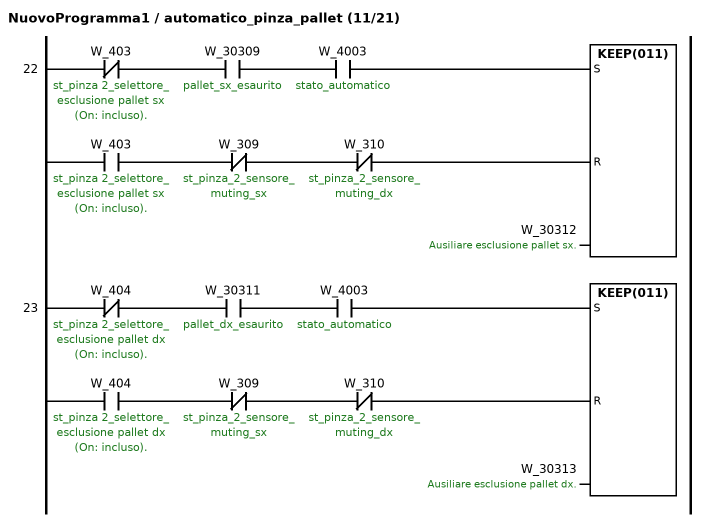
; [picture p72: NuovoProgramma1 / automatico_pinza_pallet, rungs 22-23]
; rung 22
LDNOT W_403  ; st_pinza 2_selettore_esclusione pallet sx (On: incluso).
AND W_30309  ; pallet_sx_esaurito
AND W_4003  ; stato_automatico
LD W_403  ; st_pinza 2_selettore_esclusione pallet sx (On: incluso).
ANDNOT W_309  ; st_pinza_2_sensore_muting_sx
ANDNOT W_310  ; st_pinza_2_sensore_muting_dx
KEEP(011) W_30312  ; Ausiliare esclusione pallet sx.
; rung 23
LDNOT W_404  ; st_pinza 2_selettore_esclusione pallet dx (On: incluso).
AND W_30311  ; pallet_dx_esaurito
AND W_4003  ; stato_automatico
LD W_404  ; st_pinza 2_selettore_esclusione pallet dx (On: incluso).
ANDNOT W_309  ; st_pinza_2_sensore_muting_sx
ANDNOT W_310  ; st_pinza_2_sensore_muting_dx
KEEP(011) W_30313  ; Ausiliare esclusione pallet dx.

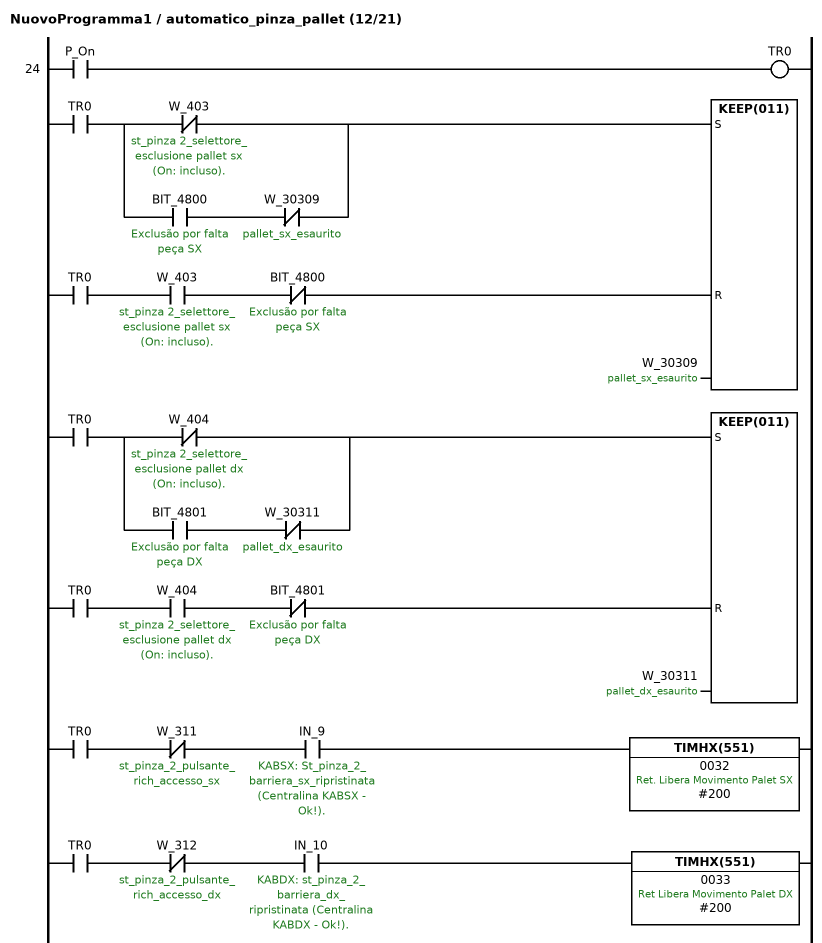

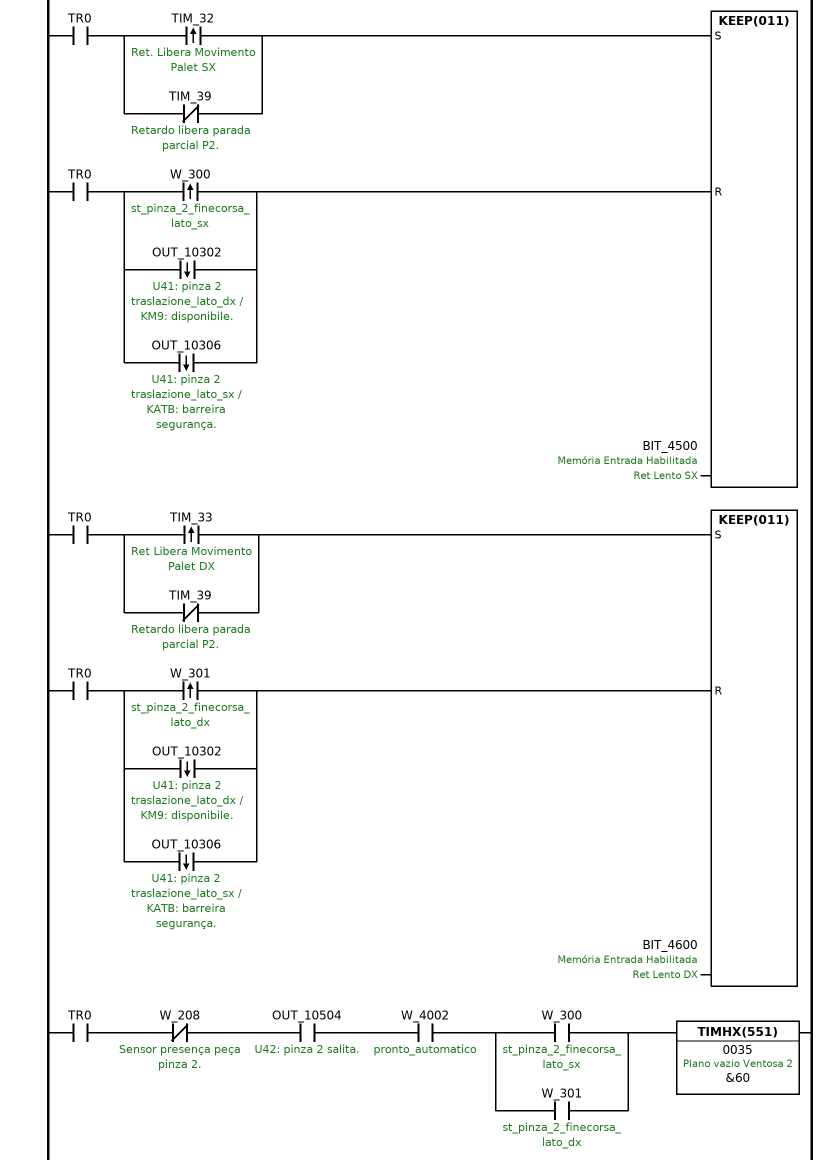

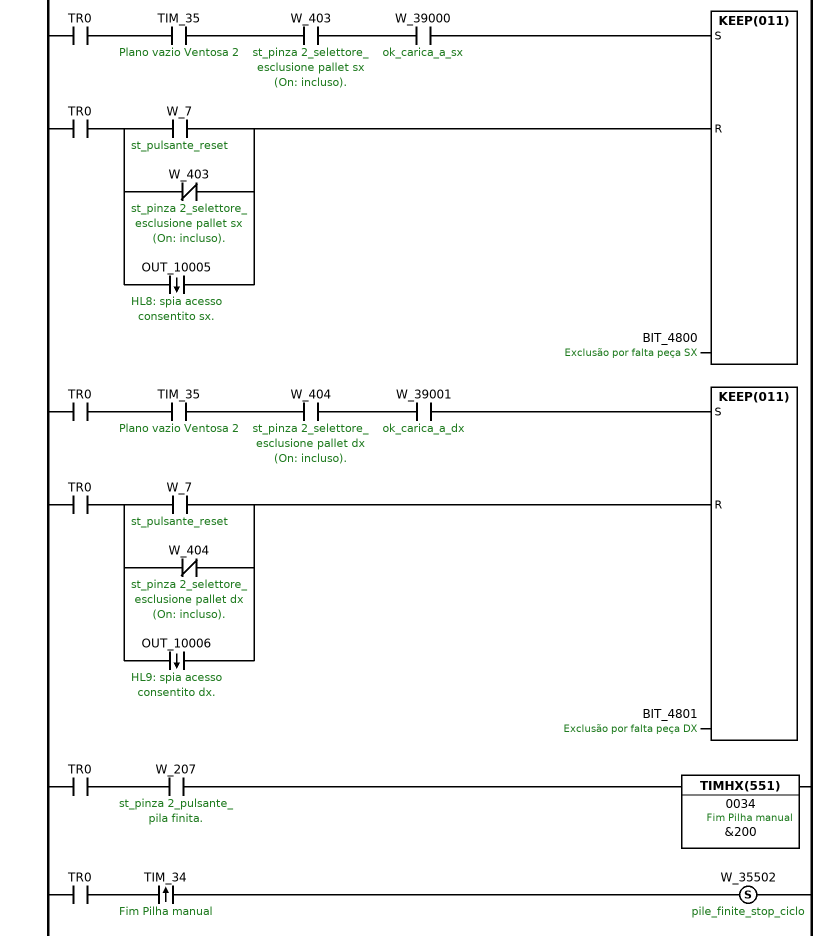
; rung 24
LD P_On
OUT TR0
LDNOT W_403  ; st_pinza 2_selettore_esclusione pallet sx (On: incluso).
LD BIT_4800  ; Exclusão por falta peça SX
ANDNOT W_30309  ; pallet_sx_esaurito
ORLD
ANDLD
LD TR0
AND W_403  ; st_pinza 2_selettore_esclusione pallet sx (On: incluso).
ANDNOT BIT_4800  ; Exclusão por falta peça SX
KEEP(011) W_30309  ; pallet_sx_esaurito
LD TR0
LDNOT W_404  ; st_pinza 2_selettore_esclusione pallet dx (On: incluso).
LD BIT_4801  ; Exclusão por falta peça DX
ANDNOT W_30311  ; pallet_dx_esaurito
ORLD
ANDLD
LD TR0
AND W_404  ; st_pinza 2_selettore_esclusione pallet dx (On: incluso).
ANDNOT BIT_4801  ; Exclusão por falta peça DX
KEEP(011) W_30311  ; pallet_dx_esaurito
LD TR0
ANDNOT W_311  ; st_pinza_2_pulsante_rich_accesso_sx
AND IN_9  ; KABSX: St_pinza_2_barriera_sx_ripristinata (Centralina KABSX - Ok!).
TIMHX(551) 0032 #200  ; Ret. Libera Movimento Palet SX
LD TR0
ANDNOT W_312  ; st_pinza_2_pulsante_rich_accesso_dx
AND IN_10  ; KABDX: st_pinza_2_barriera_dx_ripristinata (Centralina KABDX - Ok!).
TIMHX(551) 0033 #200  ; Ret Libera Movimento Palet DX
LD TR0
@LD TIM_32  ; Ret. Libera Movimento Palet SX
ORNOT TIM_39  ; Retardo libera parada parcial P2.
ANDLD
LD TR0
@LD W_300  ; st_pinza_2_finecorsa_lato_sx
%OR OUT_10302  ; U41: pinza 2 traslazione_lato_dx / KM9: disponibile.
%OR OUT_10306  ; U41: pinza 2 traslazione_lato_sx / KATB: barreira segurança.
ANDLD
KEEP(011) BIT_4500  ; Memória Entrada Habilitada Ret Lento SX
LD TR0
@LD TIM_33  ; Ret Libera Movimento Palet DX
ORNOT TIM_39  ; Retardo libera parada parcial P2.
ANDLD
LD TR0
@LD W_301  ; st_pinza_2_finecorsa_lato_dx
%OR OUT_10302  ; U41: pinza 2 traslazione_lato_dx / KM9: disponibile.
%OR OUT_10306  ; U41: pinza 2 traslazione_lato_sx / KATB: barreira segurança.
ANDLD
KEEP(011) BIT_4600  ; Memória Entrada Habilitada Ret Lento DX
LD TR0
ANDNOT W_208  ; Sensor presença peça pinza 2.
AND OUT_10504  ; U42: pinza 2 salita.
AND W_4002  ; pronto_automatico
LD W_300  ; st_pinza_2_finecorsa_lato_sx
OR W_301  ; st_pinza_2_finecorsa_lato_dx
ANDLD
TIMHX(551) 0035 &60  ; Plano vazio Ventosa 2
LD TR0
AND TIM_35  ; Plano vazio Ventosa 2
AND W_403  ; st_pinza 2_selettore_esclusione pallet sx (On: incluso).
AND W_39000  ; ok_carica_a_sx
LD TR0
LD W_7  ; st_pulsante_reset
ORNOT W_403  ; st_pinza 2_selettore_esclusione pallet sx (On: incluso).
%OR OUT_10005  ; HL8: spia acesso consentito sx.
ANDLD
KEEP(011) BIT_4800  ; Exclusão por falta peça SX
LD TR0
AND TIM_35  ; Plano vazio Ventosa 2
AND W_404  ; st_pinza 2_selettore_esclusione pallet dx (On: incluso).
AND W_39001  ; ok_carica_a_dx
LD TR0
LD W_7  ; st_pulsante_reset
ORNOT W_404  ; st_pinza 2_selettore_esclusione pallet dx (On: incluso).
%OR OUT_10006  ; HL9: spia acesso consentito dx.
ANDLD
KEEP(011) BIT_4801  ; Exclusão por falta peça DX
LD TR0
AND W_207  ; st_pinza 2_pulsante_pila finita.
TIMHX(551) 0034 &200  ; Fim Pilha manual
LD TR0
@AND TIM_34  ; Fim Pilha manual
SET W_35502  ; pile_finite_stop_ciclo

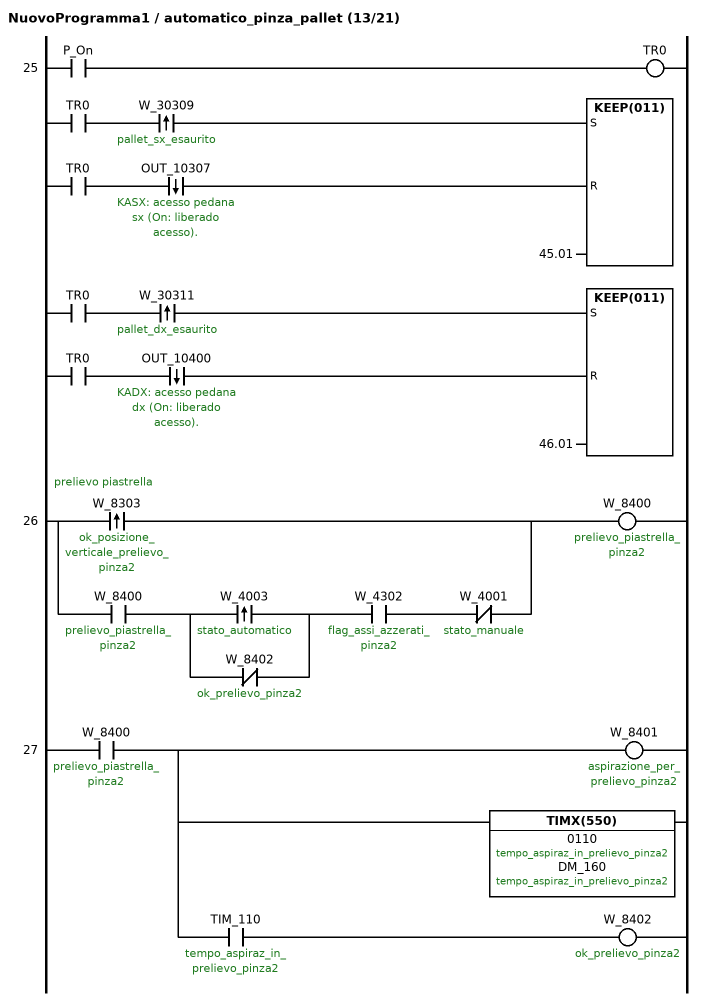
; rung 25
LD P_On
OUT TR0
@AND W_30309  ; pallet_sx_esaurito
LD TR0
%AND OUT_10307  ; KASX: acesso pedana sx (On: liberado acesso).
KEEP(011) 45.01
LD TR0
@AND W_30311  ; pallet_dx_esaurito
LD TR0
%AND OUT_10400  ; KADX: acesso pedana dx (On: liberado acesso).
KEEP(011) 46.01
; rung 26: prelievo piastrella
@LD W_8303  ; ok_posizione_verticale_prelievo_pinza2
LD W_8400  ; prelievo_piastrella_pinza2
@LD W_4003  ; stato_automatico
ORNOT W_8402  ; ok_prelievo_pinza2
ANDLD
AND W_4302  ; flag_assi_azzerati_pinza2
ANDNOT W_4001  ; stato_manuale
ORLD
OUT W_8400  ; prelievo_piastrella_pinza2
; rung 27
LD W_8400  ; prelievo_piastrella_pinza2
OUT W_8401  ; aspirazione_per_prelievo_pinza2
TIMX(550) 0110 DM_160  ; tempo_aspiraz_in_prelievo_pinza2
AND TIM_110  ; tempo_aspiraz_in_prelievo_pinza2
OUT W_8402  ; ok_prelievo_pinza2

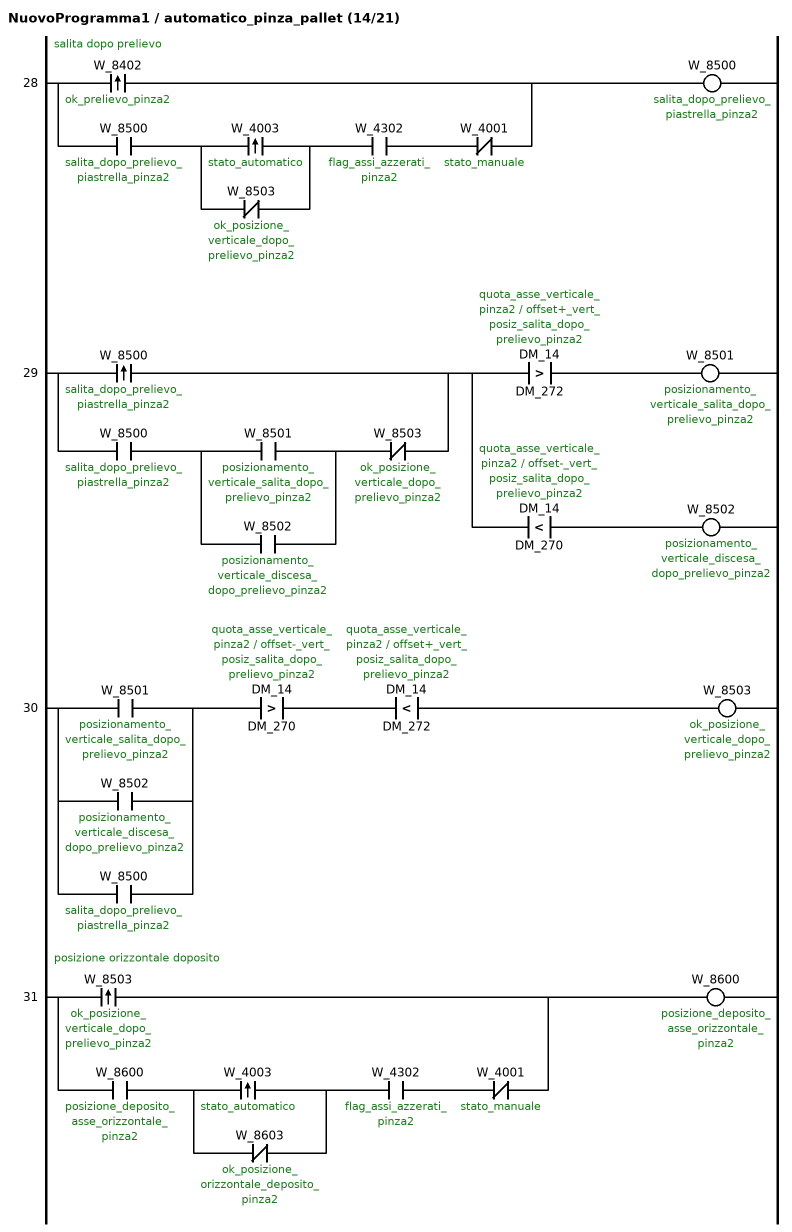
; rung 28: salita dopo prelievo
@LD W_8402  ; ok_prelievo_pinza2
LD W_8500  ; salita_dopo_prelievo_piastrella_pinza2
@LD W_4003  ; stato_automatico
ORNOT W_8503  ; ok_posizione_verticale_dopo_prelievo_pinza2
ANDLD
AND W_4302  ; flag_assi_azzerati_pinza2
ANDNOT W_4001  ; stato_manuale
ORLD
OUT W_8500  ; salita_dopo_prelievo_piastrella_pinza2
; rung 29
@LD W_8500  ; salita_dopo_prelievo_piastrella_pinza2
LD W_8500  ; salita_dopo_prelievo_piastrella_pinza2
LD W_8501  ; posizionamento_verticale_salita_dopo_prelievo_pinza2
OR W_8502  ; posizionamento_verticale_discesa_dopo_prelievo_pinza2
ANDLD
ANDNOT W_8503  ; ok_posizione_verticale_dopo_prelievo_pinza2
ORLD
OUT TR0
AND>SL(323) DM_14 DM_272  ; quota_asse_verticale_pinza2, offset+_vert_posiz_salita_dopo_prelievo_pinza2
OUT W_8501  ; posizionamento_verticale_salita_dopo_prelievo_pinza2
LD TR0
AND<SL(313) DM_14 DM_270  ; quota_asse_verticale_pinza2, offset-_vert_posiz_salita_dopo_prelievo_pinza2
OUT W_8502  ; posizionamento_verticale_discesa_dopo_prelievo_pinza2
; rung 30
LD W_8501  ; posizionamento_verticale_salita_dopo_prelievo_pinza2
OR W_8502  ; posizionamento_verticale_discesa_dopo_prelievo_pinza2
OR W_8500  ; salita_dopo_prelievo_piastrella_pinza2
AND>SL(323) DM_14 DM_270  ; quota_asse_verticale_pinza2, offset-_vert_posiz_salita_dopo_prelievo_pinza2
AND<SL(313) DM_14 DM_272  ; quota_asse_verticale_pinza2, offset+_vert_posiz_salita_dopo_prelievo_pinza2
OUT W_8503  ; ok_posizione_verticale_dopo_prelievo_pinza2
; rung 31: posizione orizzontale doposito
@LD W_8503  ; ok_posizione_verticale_dopo_prelievo_pinza2
LD W_8600  ; posizione_deposito_asse_orizzontale_pinza2
@LD W_4003  ; stato_automatico
ORNOT W_8603  ; ok_posizione_orizzontale_deposito_pinza2
ANDLD
AND W_4302  ; flag_assi_azzerati_pinza2
ANDNOT W_4001  ; stato_manuale
ORLD
OUT W_8600  ; posizione_deposito_asse_orizzontale_pinza2

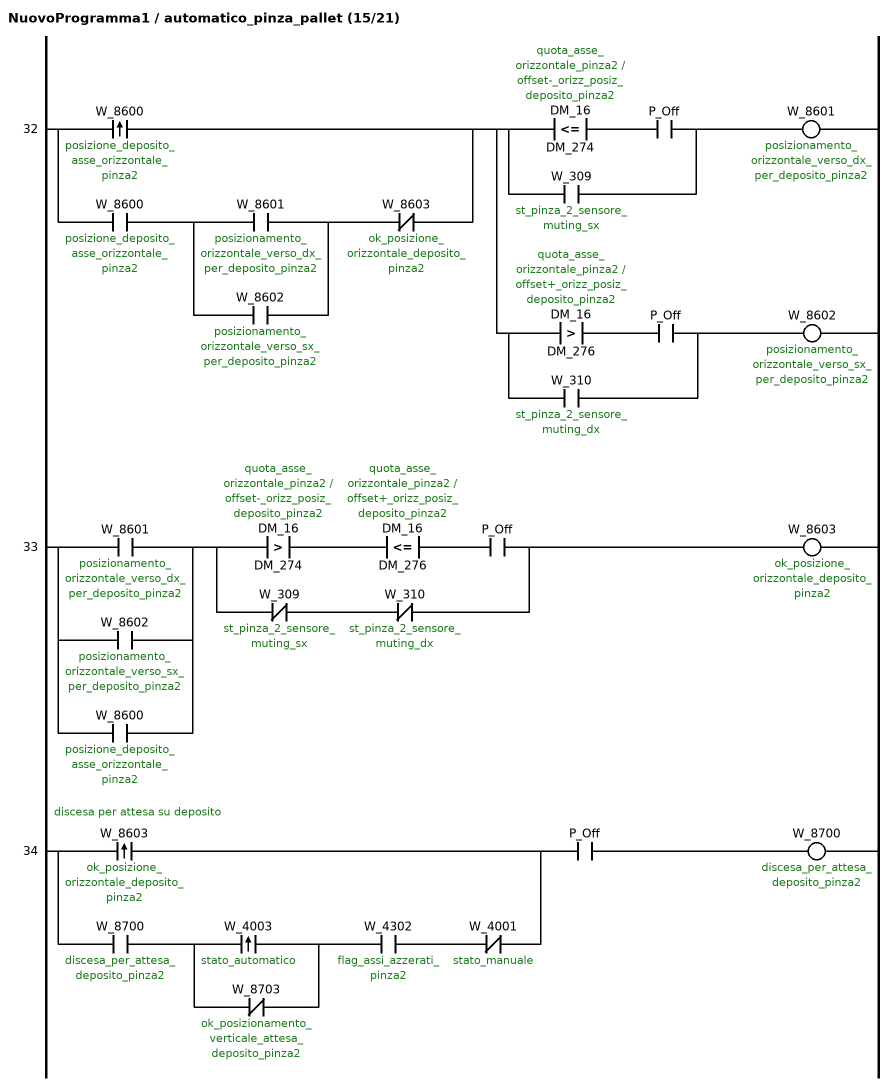
; rung 32
@LD W_8600  ; posizione_deposito_asse_orizzontale_pinza2
LD W_8600  ; posizione_deposito_asse_orizzontale_pinza2
LD W_8601  ; posizionamento_orizzontale_verso_dx_per_deposito_pinza2
OR W_8602  ; posizionamento_orizzontale_verso_sx_per_deposito_pinza2
ANDLD
ANDNOT W_8603  ; ok_posizione_orizzontale_deposito_pinza2
ORLD
OUT TR0
LD<=SL(318) DM_16 DM_274  ; quota_asse_orizzontale_pinza2, offset-_orizz_posiz_deposito_pinza2
AND P_Off
OR W_309  ; st_pinza_2_sensore_muting_sx
ANDLD
OUT W_8601  ; posizionamento_orizzontale_verso_dx_per_deposito_pinza2
LD TR0
LD>SL(323) DM_16 DM_276  ; quota_asse_orizzontale_pinza2, offset+_orizz_posiz_deposito_pinza2
AND P_Off
OR W_310  ; st_pinza_2_sensore_muting_dx
ANDLD
OUT W_8602  ; posizionamento_orizzontale_verso_sx_per_deposito_pinza2
; rung 33
LD W_8601  ; posizionamento_orizzontale_verso_dx_per_deposito_pinza2
OR W_8602  ; posizionamento_orizzontale_verso_sx_per_deposito_pinza2
OR W_8600  ; posizione_deposito_asse_orizzontale_pinza2
LD>SL(323) DM_16 DM_274  ; quota_asse_orizzontale_pinza2, offset-_orizz_posiz_deposito_pinza2
AND<=SL(318) DM_16 DM_276  ; quota_asse_orizzontale_pinza2, offset+_orizz_posiz_deposito_pinza2
AND P_Off
LDNOT W_309  ; st_pinza_2_sensore_muting_sx
ANDNOT W_310  ; st_pinza_2_sensore_muting_dx
ORLD
ANDLD
OUT W_8603  ; ok_posizione_orizzontale_deposito_pinza2
; rung 34: discesa per attesa su deposito
@LD W_8603  ; ok_posizione_orizzontale_deposito_pinza2
LD W_8700  ; discesa_per_attesa_deposito_pinza2
@LD W_4003  ; stato_automatico
ORNOT W_8703  ; ok_posizionamento_verticale_attesa_deposito_pinza2
ANDLD
AND W_4302  ; flag_assi_azzerati_pinza2
ANDNOT W_4001  ; stato_manuale
ORLD
AND P_Off
OUT W_8700  ; discesa_per_attesa_deposito_pinza2

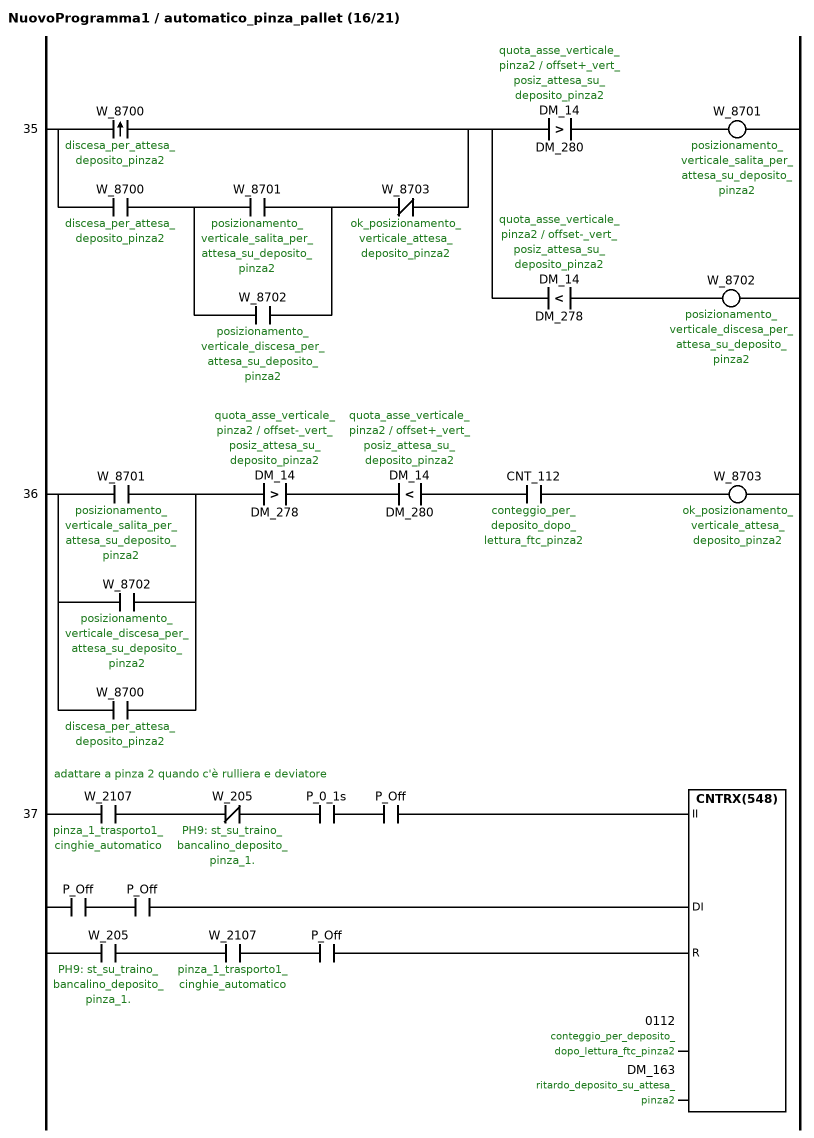
; rung 35
@LD W_8700  ; discesa_per_attesa_deposito_pinza2
LD W_8700  ; discesa_per_attesa_deposito_pinza2
LD W_8701  ; posizionamento_verticale_salita_per_attesa_su_deposito_pinza2
OR W_8702  ; posizionamento_verticale_discesa_per_attesa_su_deposito_pinza2
ANDLD
ANDNOT W_8703  ; ok_posizionamento_verticale_attesa_deposito_pinza2
ORLD
OUT TR0
AND>SL(323) DM_14 DM_280  ; quota_asse_verticale_pinza2, offset+_vert_posiz_attesa_su_deposito_pinza2
OUT W_8701  ; posizionamento_verticale_salita_per_attesa_su_deposito_pinza2
LD TR0
AND<SL(313) DM_14 DM_278  ; quota_asse_verticale_pinza2, offset-_vert_posiz_attesa_su_deposito_pinza2
OUT W_8702  ; posizionamento_verticale_discesa_per_attesa_su_deposito_pinza2
; rung 36
LD W_8701  ; posizionamento_verticale_salita_per_attesa_su_deposito_pinza2
OR W_8702  ; posizionamento_verticale_discesa_per_attesa_su_deposito_pinza2
OR W_8700  ; discesa_per_attesa_deposito_pinza2
AND>SL(323) DM_14 DM_278  ; quota_asse_verticale_pinza2, offset-_vert_posiz_attesa_su_deposito_pinza2
AND<SL(313) DM_14 DM_280  ; quota_asse_verticale_pinza2, offset+_vert_posiz_attesa_su_deposito_pinza2
AND CNT_112  ; conteggio_per_deposito_dopo_lettura_ftc_pinza2
OUT W_8703  ; ok_posizionamento_verticale_attesa_deposito_pinza2
; rung 37: adattare a pinza 2 quando c'è rulliera e deviatore
LD W_2107  ; pinza_1_trasporto1_cinghie_automatico
ANDNOT W_205  ; PH9: st_su_traino_bancalino_deposito_pinza_1.
AND P_0_1s
AND P_Off
LD P_Off
AND P_Off
LD W_205  ; PH9: st_su_traino_bancalino_deposito_pinza_1.
AND W_2107  ; pinza_1_trasporto1_cinghie_automatico
AND P_Off
CNTRX(548) 0112 DM_163  ; ritardo_deposito_su_attesa_pinza2, conteggio_per_deposito_dopo_lettura_ftc_pinza2

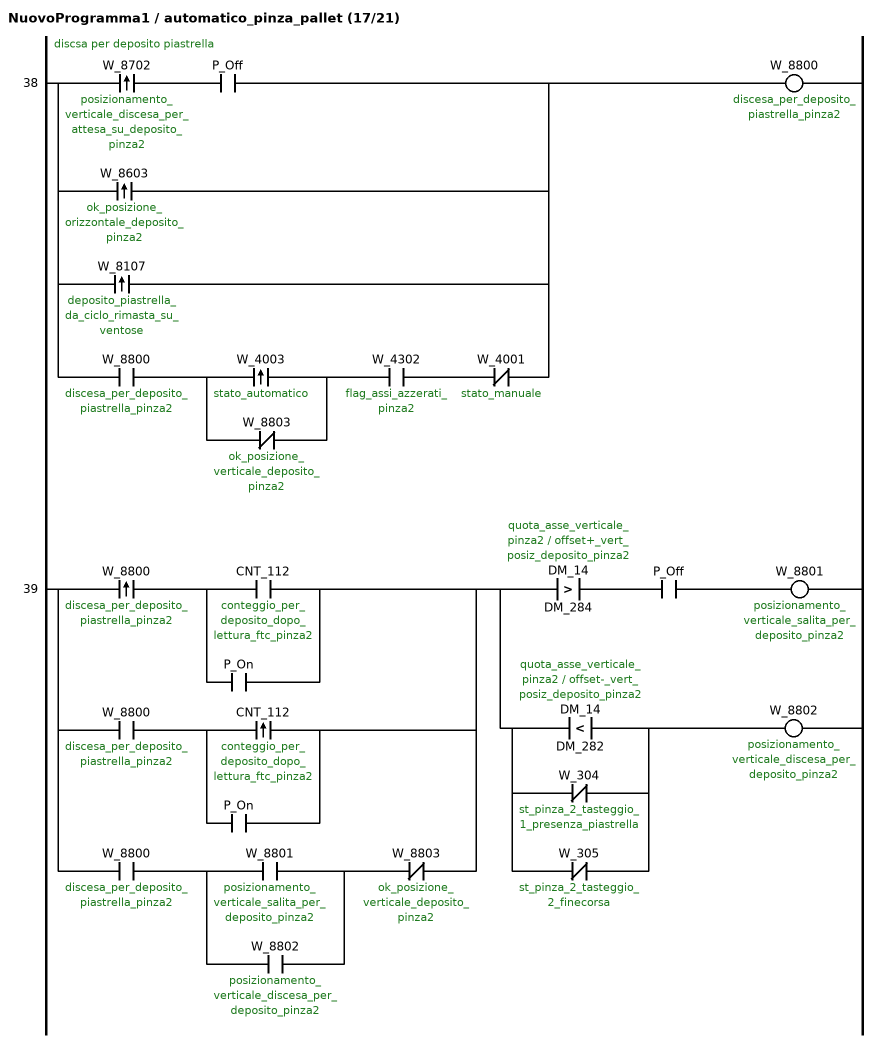
; rung 38: discsa per deposito piastrella
@LD W_8702  ; posizionamento_verticale_discesa_per_attesa_su_deposito_pinza2
AND P_Off
@OR W_8603  ; ok_posizione_orizzontale_deposito_pinza2
@OR W_8107  ; deposito_piastrella_da_ciclo_rimasta_su_ventose
LD W_8800  ; discesa_per_deposito_piastrella_pinza2
@LD W_4003  ; stato_automatico
ORNOT W_8803  ; ok_posizione_verticale_deposito_pinza2
ANDLD
AND W_4302  ; flag_assi_azzerati_pinza2
ANDNOT W_4001  ; stato_manuale
ORLD
OUT W_8800  ; discesa_per_deposito_piastrella_pinza2
; rung 39
@LD W_8800  ; discesa_per_deposito_piastrella_pinza2
LD CNT_112  ; conteggio_per_deposito_dopo_lettura_ftc_pinza2
OR P_On
ANDLD
LD W_8800  ; discesa_per_deposito_piastrella_pinza2
@LD CNT_112  ; conteggio_per_deposito_dopo_lettura_ftc_pinza2
OR P_On
ANDLD
ORLD
LD W_8800  ; discesa_per_deposito_piastrella_pinza2
LD W_8801  ; posizionamento_verticale_salita_per_deposito_pinza2
OR W_8802  ; posizionamento_verticale_discesa_per_deposito_pinza2
ANDLD
ANDNOT W_8803  ; ok_posizione_verticale_deposito_pinza2
ORLD
OUT TR0
AND>SL(323) DM_14 DM_284  ; quota_asse_verticale_pinza2, offset+_vert_posiz_deposito_pinza2
AND P_Off
OUT W_8801  ; posizionamento_verticale_salita_per_deposito_pinza2
LD TR0
LD<SL(313) DM_14 DM_282  ; quota_asse_verticale_pinza2, offset-_vert_posiz_deposito_pinza2
ORNOT W_304  ; st_pinza_2_tasteggio_1_presenza_piastrella
ORNOT W_305  ; st_pinza_2_tasteggio_2_finecorsa
ANDLD
OUT W_8802  ; posizionamento_verticale_discesa_per_deposito_pinza2

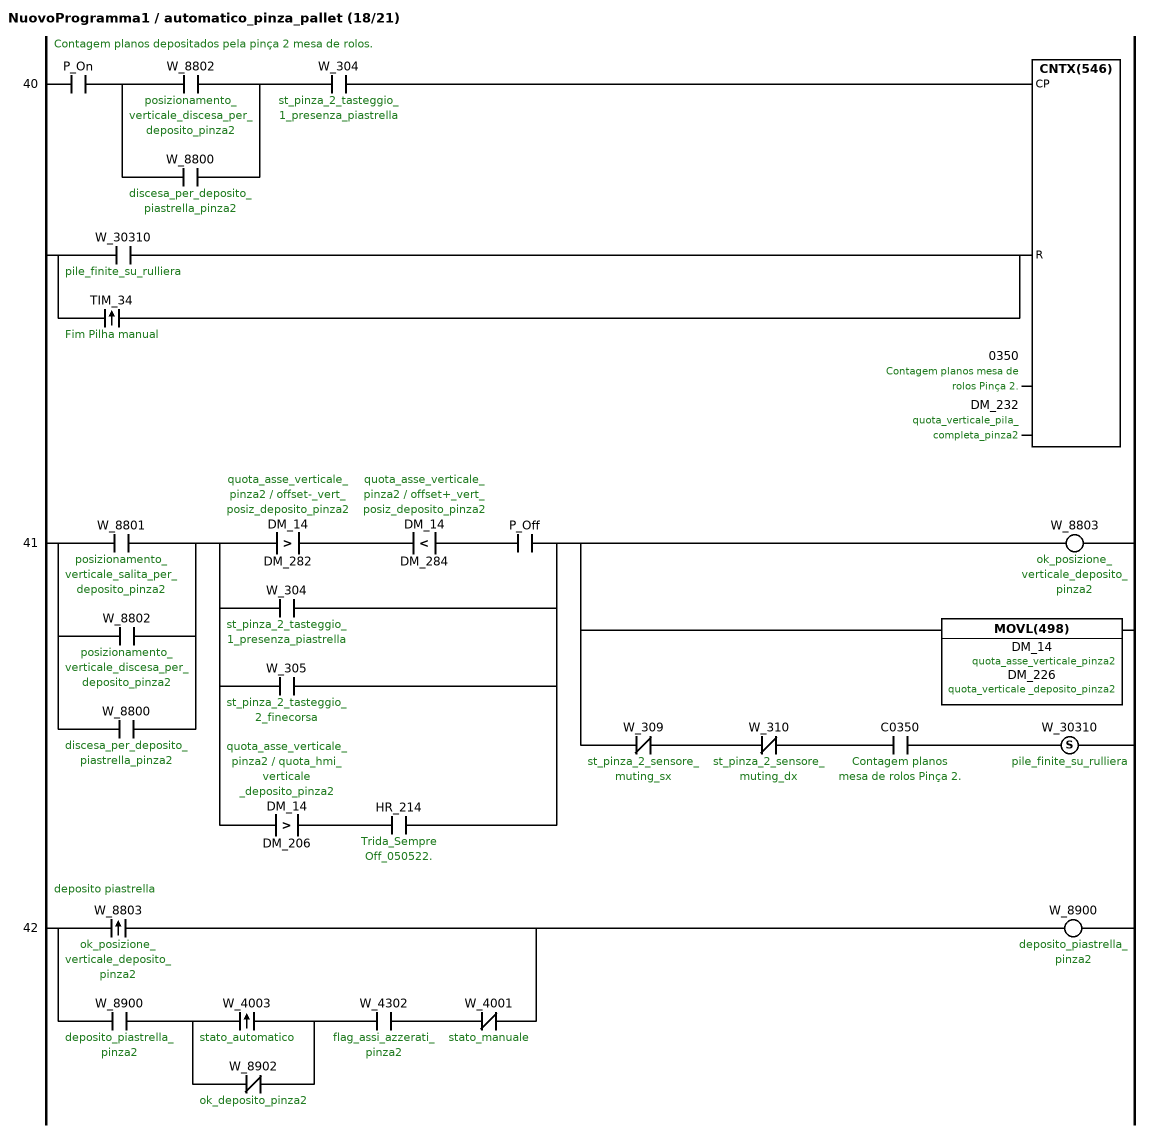
; rung 40: Contagem planos depositados pela pinça 2 mesa de rolos.
LD P_On
LD W_8802  ; posizionamento_verticale_discesa_per_deposito_pinza2
OR W_8800  ; discesa_per_deposito_piastrella_pinza2
ANDLD
AND W_304  ; st_pinza_2_tasteggio_1_presenza_piastrella
LD W_30310  ; pile_finite_su_rulliera
@OR TIM_34  ; Fim Pilha manual
CNTX(546) 0350 DM_232  ; quota_verticale_pila_completa_pinza2, Contagem planos mesa de rolos Pinça 2.
; rung 41
LD W_8801  ; posizionamento_verticale_salita_per_deposito_pinza2
OR W_8802  ; posizionamento_verticale_discesa_per_deposito_pinza2
OR W_8800  ; discesa_per_deposito_piastrella_pinza2
LD>SL(323) DM_14 DM_282  ; quota_asse_verticale_pinza2, offset-_vert_posiz_deposito_pinza2
AND<SL(313) DM_14 DM_284  ; quota_asse_verticale_pinza2, offset+_vert_posiz_deposito_pinza2
AND P_Off
OR W_304  ; st_pinza_2_tasteggio_1_presenza_piastrella
OR W_305  ; st_pinza_2_tasteggio_2_finecorsa
LD>SL(323) DM_14 DM_206  ; quota_asse_verticale_pinza2, quota_hmi_verticale _deposito_pinza2
AND HR_214  ; Trida_Sempre Off_050522.
ORLD
ANDLD
OUT W_8803  ; ok_posizione_verticale_deposito_pinza2
MOVL(498) DM_14 DM_226  ; quota_asse_verticale_pinza2, quota_verticale _deposito_pinza2
ANDNOT W_309  ; st_pinza_2_sensore_muting_sx
ANDNOT W_310  ; st_pinza_2_sensore_muting_dx
AND C0350  ; Contagem planos mesa de rolos Pinça 2.
SET W_30310  ; pile_finite_su_rulliera
; rung 42: deposito piastrella
@LD W_8803  ; ok_posizione_verticale_deposito_pinza2
LD W_8900  ; deposito_piastrella_pinza2
@LD W_4003  ; stato_automatico
ORNOT W_8902  ; ok_deposito_pinza2
ANDLD
AND W_4302  ; flag_assi_azzerati_pinza2
ANDNOT W_4001  ; stato_manuale
ORLD
OUT W_8900  ; deposito_piastrella_pinza2

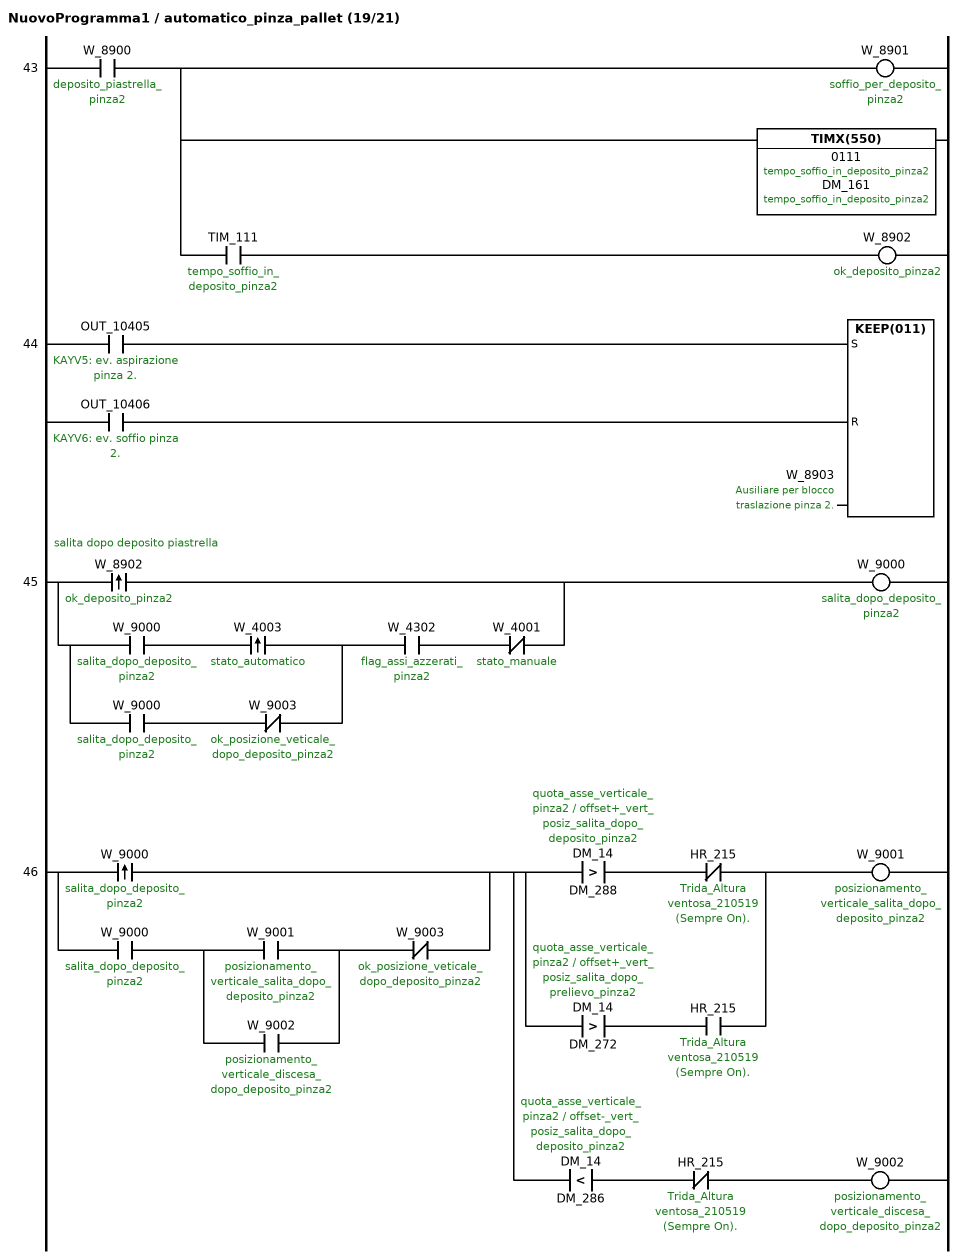
; rung 43
LD W_8900  ; deposito_piastrella_pinza2
OUT W_8901  ; soffio_per_deposito_pinza2
TIMX(550) 0111 DM_161  ; tempo_soffio_in_deposito_pinza2
AND TIM_111  ; tempo_soffio_in_deposito_pinza2
OUT W_8902  ; ok_deposito_pinza2
; rung 44
LD OUT_10405  ; KAYV5: ev. aspirazione pinza 2.
LD OUT_10406  ; KAYV6: ev. soffio pinza 2.
KEEP(011) W_8903  ; Ausiliare per blocco traslazione pinza 2.
; rung 45: salita dopo deposito piastrella
@LD W_8902  ; ok_deposito_pinza2
LD W_9000  ; salita_dopo_deposito_pinza2
@AND W_4003  ; stato_automatico
LD W_9000  ; salita_dopo_deposito_pinza2
ANDNOT W_9003  ; ok_posizione_veticale_dopo_deposito_pinza2
ORLD
AND W_4302  ; flag_assi_azzerati_pinza2
ANDNOT W_4001  ; stato_manuale
ORLD
OUT W_9000  ; salita_dopo_deposito_pinza2
; rung 46
@LD W_9000  ; salita_dopo_deposito_pinza2
LD W_9000  ; salita_dopo_deposito_pinza2
LD W_9001  ; posizionamento_verticale_salita_dopo_deposito_pinza2
OR W_9002  ; posizionamento_verticale_discesa_dopo_deposito_pinza2
ANDLD
ANDNOT W_9003  ; ok_posizione_veticale_dopo_deposito_pinza2
ORLD
OUT TR0
LD>SL(323) DM_14 DM_288  ; quota_asse_verticale_pinza2, offset+_vert_posiz_salita_dopo_deposito_pinza2
ANDNOT HR_215  ; Trida_Altura ventosa_210519 (Sempre On).  // HR 2.15: Modificado para ventosa subir vazia no centro até a altura da translação com ventosa carregada. / (Para evitar bater no pancone). / 210519. / .
LD>SL(323) DM_14 DM_272  ; quota_asse_verticale_pinza2, offset+_vert_posiz_salita_dopo_prelievo_pinza2
AND HR_215  ; Trida_Altura ventosa_210519 (Sempre On).  // HR 2.15: Modificado para ventosa subir vazia no centro até a altura da translação com ventosa carregada. / (Para evitar bater no pancone). / 210519. / .
ORLD
ANDLD
OUT W_9001  ; posizionamento_verticale_salita_dopo_deposito_pinza2
LD TR0
AND<SL(313) DM_14 DM_286  ; quota_asse_verticale_pinza2, offset-_vert_posiz_salita_dopo_deposito_pinza2
ANDNOT HR_215  ; Trida_Altura ventosa_210519 (Sempre On).
OUT W_9002  ; posizionamento_verticale_discesa_dopo_deposito_pinza2

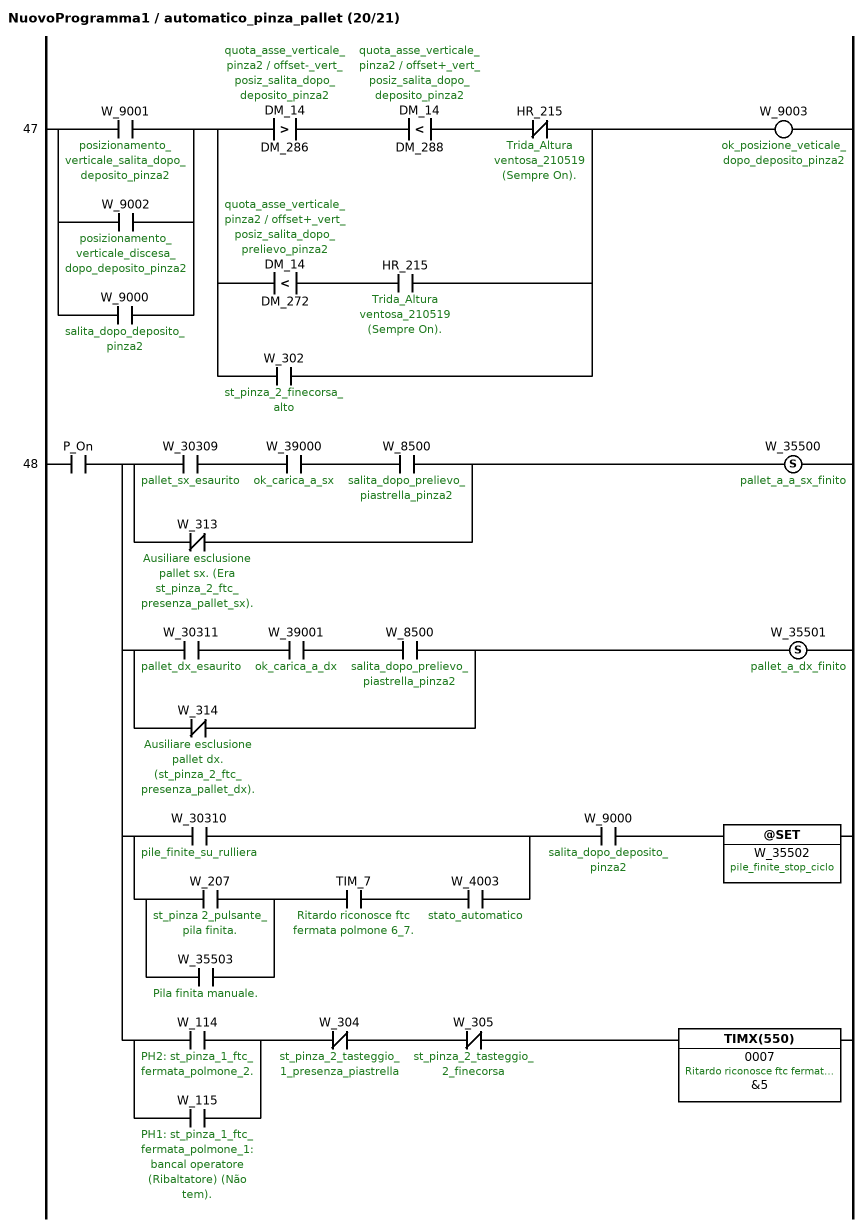
; rung 47
LD W_9001  ; posizionamento_verticale_salita_dopo_deposito_pinza2
OR W_9002  ; posizionamento_verticale_discesa_dopo_deposito_pinza2
OR W_9000  ; salita_dopo_deposito_pinza2
LD>SL(323) DM_14 DM_286  ; quota_asse_verticale_pinza2, offset-_vert_posiz_salita_dopo_deposito_pinza2
AND<SL(313) DM_14 DM_288  ; quota_asse_verticale_pinza2, offset+_vert_posiz_salita_dopo_deposito_pinza2
ANDNOT HR_215  ; Trida_Altura ventosa_210519 (Sempre On).  // HR 2.15: Modificado para ventosa subir vazia no centro até a altura da translação com ventosa carregada. / (Para evitar bater no pancone). / 210519. / .
LD<SL(313) DM_14 DM_272  ; quota_asse_verticale_pinza2, offset+_vert_posiz_salita_dopo_prelievo_pinza2
AND HR_215  ; Trida_Altura ventosa_210519 (Sempre On).  // HR 2.15: Modificado para ventosa subir vazia no centro até a altura da translação com ventosa carregada. / (Para evitar bater no pancone). / 210519. / .
ORLD
OR W_302  ; st_pinza_2_finecorsa_alto
ANDLD
OUT W_9003  ; ok_posizione_veticale_dopo_deposito_pinza2
; rung 48
LD P_On
OUT TR0
LD W_30309  ; pallet_sx_esaurito
AND W_39000  ; ok_carica_a_sx
AND W_8500  ; salita_dopo_prelievo_piastrella_pinza2
ORNOT W_313  ; Ausiliare esclusione pallet sx. (Era st_pinza_2_ftc_presenza_pallet_sx).
ANDLD
SET W_35500  ; pallet_a_a_sx_finito
LD TR0
LD W_30311  ; pallet_dx_esaurito
AND W_39001  ; ok_carica_a_dx
AND W_8500  ; salita_dopo_prelievo_piastrella_pinza2
ORNOT W_314  ; Ausiliare esclusione pallet dx. (st_pinza_2_ftc_presenza_pallet_dx).
ANDLD
SET W_35501  ; pallet_a_dx_finito
LD TR0
LD W_30310  ; pile_finite_su_rulliera
LD W_207  ; st_pinza 2_pulsante_pila finita.
OR W_35503  ; Pila finita manuale.
AND TIM_7  ; Ritardo riconosce ftc fermata polmone 6_7.
AND W_4003  ; stato_automatico
ORLD
ANDLD
AND W_9000  ; salita_dopo_deposito_pinza2
@SET W_35502  ; pile_finite_stop_ciclo
LD TR0
LD W_114  ; PH2: st_pinza_1_ftc_fermata_polmone_2.
OR W_115  ; PH1: st_pinza_1_ftc_fermata_polmone_1: bancal operatore (Ribaltatore) (Não tem).
ANDLD
ANDNOT W_304  ; st_pinza_2_tasteggio_1_presenza_piastrella
ANDNOT W_305  ; st_pinza_2_tasteggio_2_finecorsa
TIMX(550) 0007 &5  ; Ritardo riconosce ftc fermata polmone 6_7.

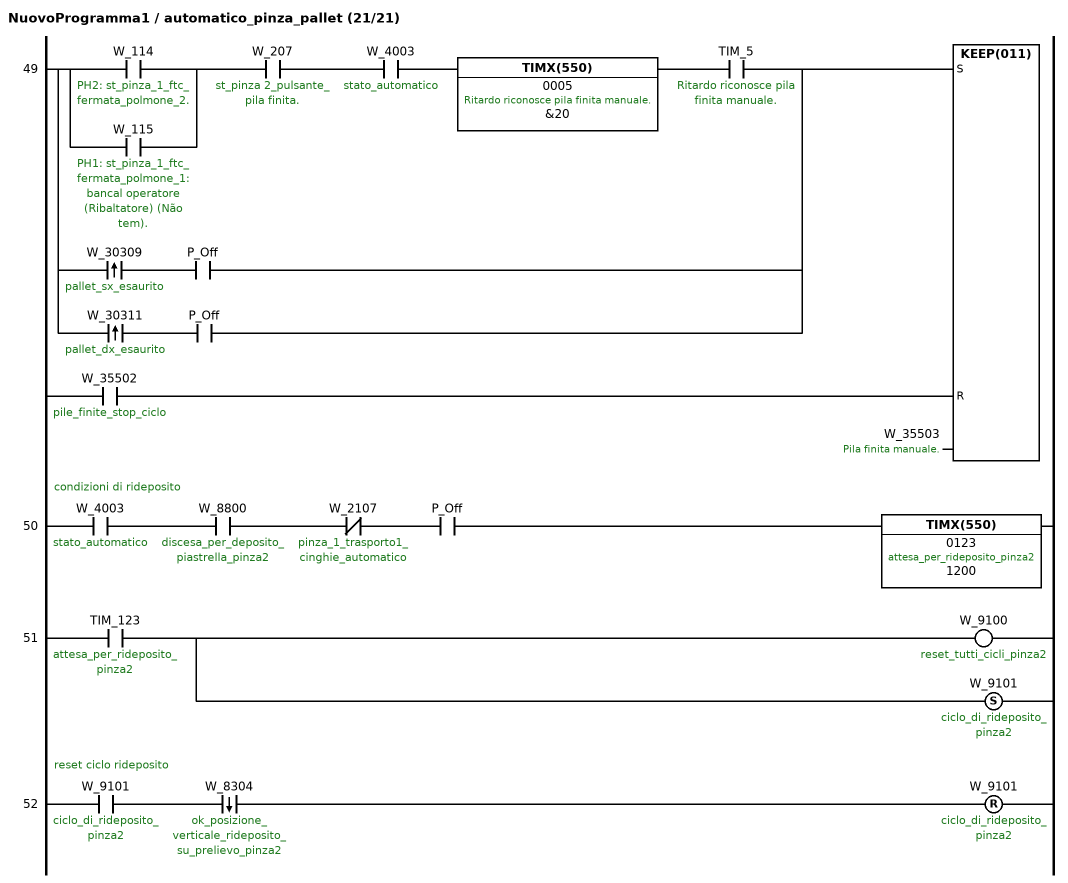
; rung 49
LD W_114  ; PH2: st_pinza_1_ftc_fermata_polmone_2.
OR W_115  ; PH1: st_pinza_1_ftc_fermata_polmone_1: bancal operatore (Ribaltatore) (Não tem).
AND W_207  ; st_pinza 2_pulsante_pila finita.
AND W_4003  ; stato_automatico
TIMX(550) 0005 &20  ; Ritardo riconosce pila finita manuale.
AND TIM_5  ; Ritardo riconosce pila finita manuale.
@LD W_30309  ; pallet_sx_esaurito
AND P_Off
@LD W_30311  ; pallet_dx_esaurito
AND P_Off
ORLD
ORLD
LD W_35502  ; pile_finite_stop_ciclo
KEEP(011) W_35503  ; Pila finita manuale.
; rung 50: condizioni di rideposito
LD W_4003  ; stato_automatico
AND W_8800  ; discesa_per_deposito_piastrella_pinza2
ANDNOT W_2107  ; pinza_1_trasporto1_cinghie_automatico
AND P_Off
TIMX(550) 0123 1200  ; attesa_per_rideposito_pinza2
; rung 51
LD TIM_123  ; attesa_per_rideposito_pinza2
OUT W_9100  ; reset_tutti_cicli_pinza2
SET W_9101  ; ciclo_di_rideposito_pinza2
; rung 52: reset ciclo rideposito
LD W_9101  ; ciclo_di_rideposito_pinza2
%AND W_8304  ; ok_posizione_verticale_rideposito_su_prelievo_pinza2
RSET W_9101  ; ciclo_di_rideposito_pinza2

### Section quote_pinza_ribaltino

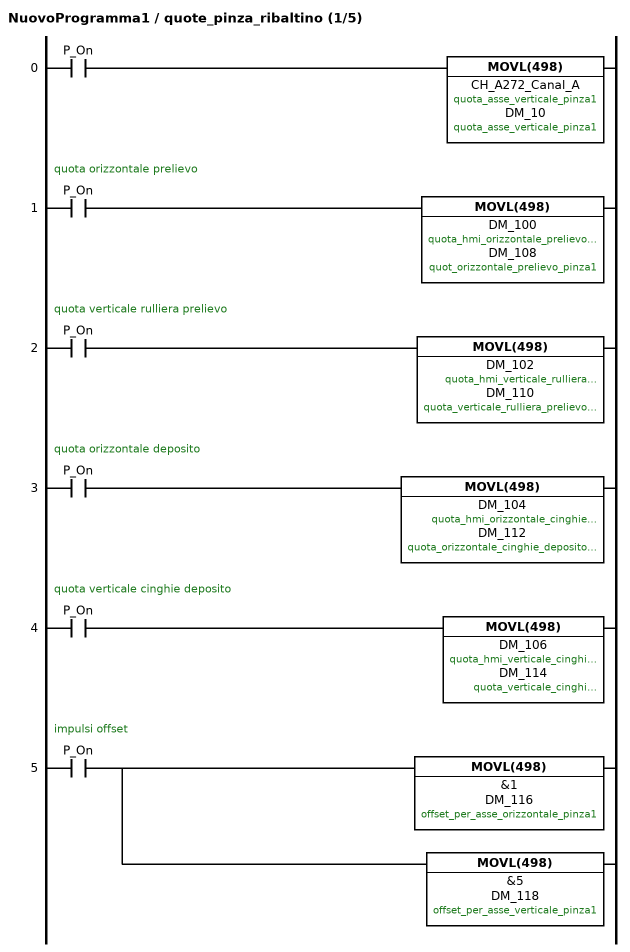
; rung 0
LD P_On
MOVL(498) CH_A272_Canal_A DM_10  ; quota_asse_verticale_pinza1
; rung 1: quota orizzontale prelievo
LD P_On
MOVL(498) DM_100 DM_108  ; quota_hmi_orizzontale_prelievo_pinza1, quot_orizzontale_prelievo_pinza1
; rung 2: quota verticale rulliera prelievo
LD P_On
MOVL(498) DM_102 DM_110  ; quota_hmi_verticale_rulliera_prelievo_pinza1, quota_verticale_rulliera_prelievo_pinza1
; rung 3: quota orizzontale deposito
LD P_On
MOVL(498) DM_104 DM_112  ; quota_hmi_orizzontale_cinghie_deposito_pinza1, quota_orizzontale_cinghie_deposito_pinza1
; rung 4: quota verticale cinghie deposito
LD P_On
MOVL(498) DM_106 DM_114  ; quota_hmi_verticale_cinghie _deposito_pinza1, quota_verticale_cinghie _deposito_pinza1
; rung 5: impulsi offset
LD P_On
MOVL(498) &1 DM_116  ; offset_per_asse_orizzontale_pinza1
MOVL(498) &5 DM_118  ; offset_per_asse_verticale_pinza1

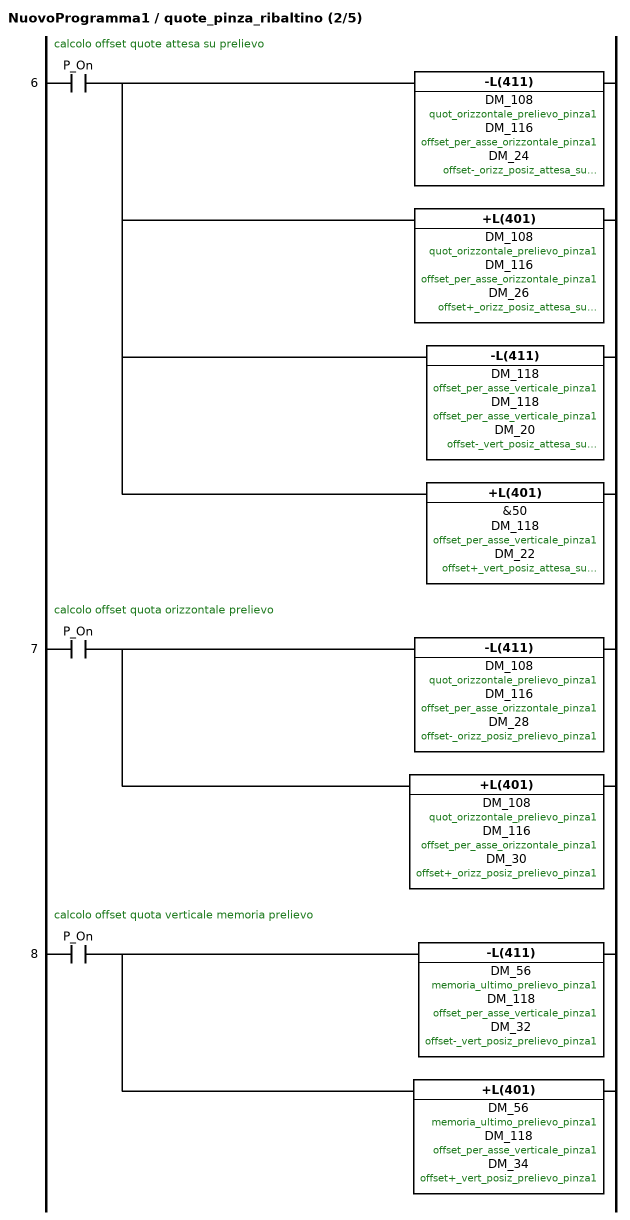
; rung 6: calcolo offset quote attesa su prelievo
LD P_On
-L(411) DM_108 DM_116 DM_24  ; quot_orizzontale_prelievo_pinza1, offset_per_asse_orizzontale_pinza1, offset-_orizz_posiz_attesa_su_prelievo_pinza1
+L(401) DM_108 DM_116 DM_26  ; quot_orizzontale_prelievo_pinza1, offset_per_asse_orizzontale_pinza1, offset+_orizz_posiz_attesa_su_prelievo_pinza1
-L(411) DM_118 DM_118 DM_20  ; offset_per_asse_verticale_pinza1, offset-_vert_posiz_attesa_su_prelievo_pinza1
+L(401) &50 DM_118 DM_22  ; offset_per_asse_verticale_pinza1, offset+_vert_posiz_attesa_su_prelievo_pinza1
; rung 7: calcolo offset quota orizzontale prelievo
LD P_On
-L(411) DM_108 DM_116 DM_28  ; quot_orizzontale_prelievo_pinza1, offset_per_asse_orizzontale_pinza1, offset-_orizz_posiz_prelievo_pinza1
+L(401) DM_108 DM_116 DM_30  ; quot_orizzontale_prelievo_pinza1, offset_per_asse_orizzontale_pinza1, offset+_orizz_posiz_prelievo_pinza1
; rung 8: calcolo offset quota verticale memoria prelievo
LD P_On
-L(411) DM_56 DM_118 DM_32  ; memoria_ultimo_prelievo_pinza1, offset_per_asse_verticale_pinza1, offset-_vert_posiz_prelievo_pinza1
+L(401) DM_56 DM_118 DM_34  ; memoria_ultimo_prelievo_pinza1, offset_per_asse_verticale_pinza1, offset+_vert_posiz_prelievo_pinza1

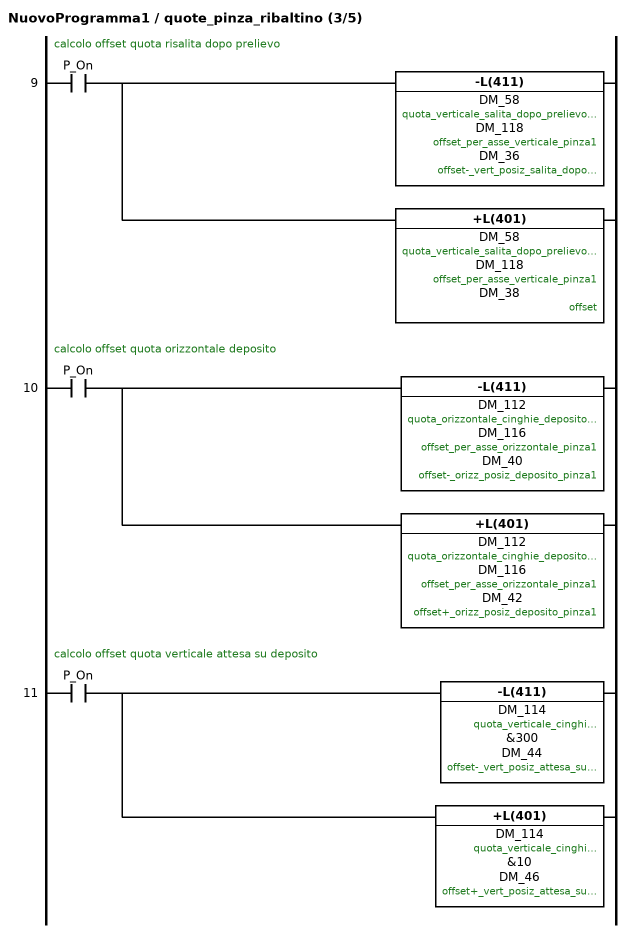
; rung 9: calcolo offset quota risalita dopo prelievo
LD P_On
-L(411) DM_58 DM_118 DM_36  ; quota_verticale_salita_dopo_prelievo_pinza1, offset_per_asse_verticale_pinza1, offset-_vert_posiz_salita_dopo_prelievo_pinza1
+L(401) DM_58 DM_118 DM_38  ; quota_verticale_salita_dopo_prelievo_pinza1, offset_per_asse_verticale_pinza1, offset
; rung 10: calcolo offset quota orizzontale deposito
LD P_On
-L(411) DM_112 DM_116 DM_40  ; quota_orizzontale_cinghie_deposito_pinza1, offset_per_asse_orizzontale_pinza1, offset-_orizz_posiz_deposito_pinza1
+L(401) DM_112 DM_116 DM_42  ; quota_orizzontale_cinghie_deposito_pinza1, offset_per_asse_orizzontale_pinza1, offset+_orizz_posiz_deposito_pinza1
; rung 11: calcolo offset quota verticale attesa su deposito
LD P_On
-L(411) DM_114 &300 DM_44  ; quota_verticale_cinghie _deposito_pinza1, offset-_vert_posiz_attesa_su_deposito_pinza1
+L(401) DM_114 &10 DM_46  ; quota_verticale_cinghie _deposito_pinza1, offset+_vert_posiz_attesa_su_deposito_pinza1

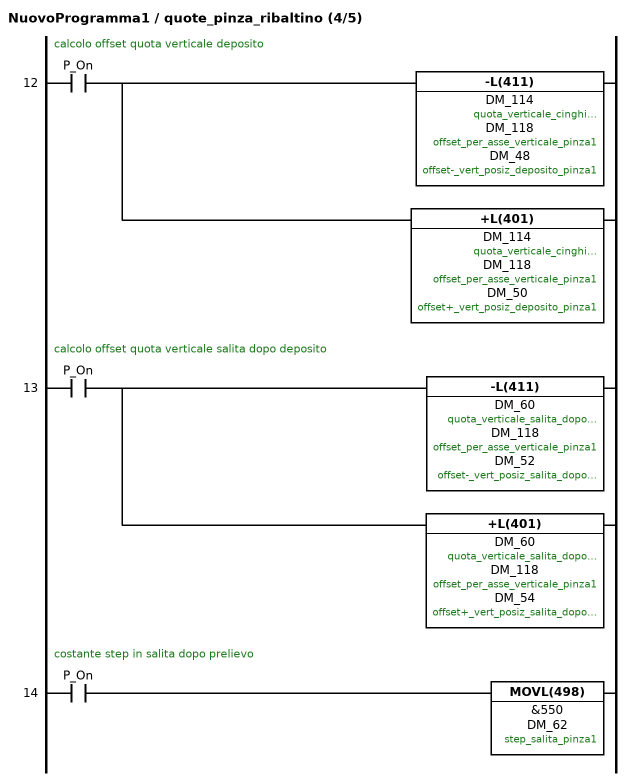
; rung 12: calcolo offset quota verticale deposito
LD P_On
-L(411) DM_114 DM_118 DM_48  ; quota_verticale_cinghie _deposito_pinza1, offset_per_asse_verticale_pinza1, offset-_vert_posiz_deposito_pinza1
+L(401) DM_114 DM_118 DM_50  ; quota_verticale_cinghie _deposito_pinza1, offset_per_asse_verticale_pinza1, offset+_vert_posiz_deposito_pinza1
; rung 13: calcolo offset quota verticale salita dopo deposito
LD P_On
-L(411) DM_60 DM_118 DM_52  ; quota_verticale_salita_dopo_deposito_pinza1, offset_per_asse_verticale_pinza1, offset-_vert_posiz_salita_dopo_deposito_pinza1
+L(401) DM_60 DM_118 DM_54  ; quota_verticale_salita_dopo_deposito_pinza1, offset_per_asse_verticale_pinza1, offset+_vert_posiz_salita_dopo_deposito_pinza1
; rung 14: costante step in salita dopo prelievo
LD P_On
MOVL(498) &550 DM_62  ; step_salita_pinza1

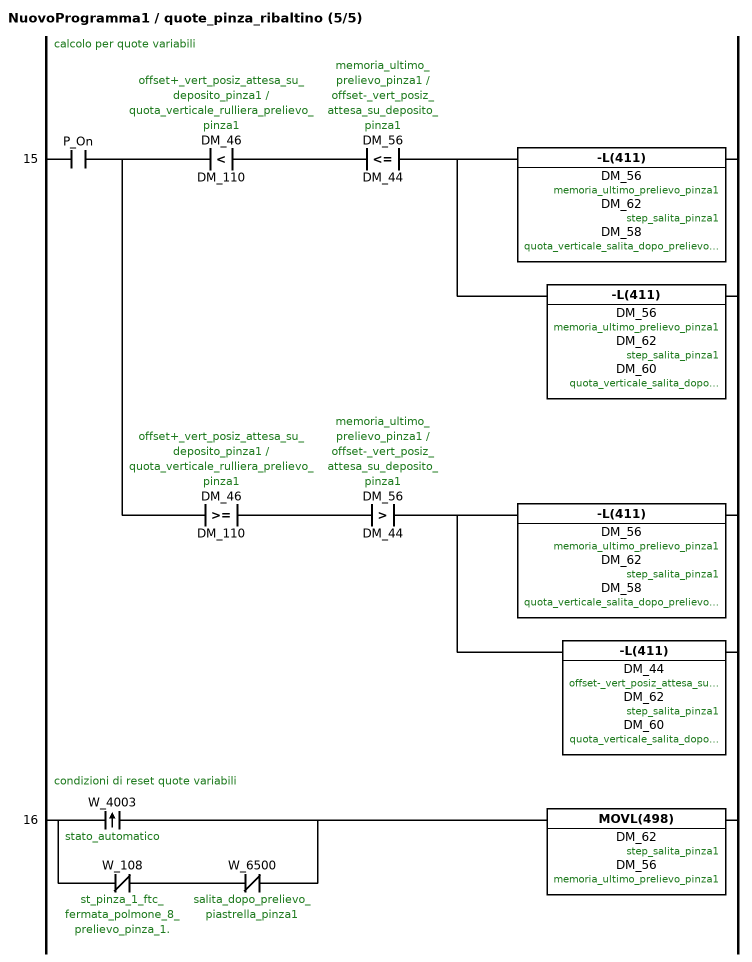
; rung 15: calcolo per quote variabili
LD P_On
OUT TR0
AND<SL(313) DM_46 DM_110  ; offset+_vert_posiz_attesa_su_deposito_pinza1, quota_verticale_rulliera_prelievo_pinza1
AND<=SL(318) DM_56 DM_44  ; memoria_ultimo_prelievo_pinza1, offset-_vert_posiz_attesa_su_deposito_pinza1
-L(411) DM_56 DM_62 DM_58  ; memoria_ultimo_prelievo_pinza1, step_salita_pinza1, quota_verticale_salita_dopo_prelievo_pinza1
-L(411) DM_56 DM_62 DM_60  ; memoria_ultimo_prelievo_pinza1, step_salita_pinza1, quota_verticale_salita_dopo_deposito_pinza1
LD TR0
AND>=SL(328) DM_46 DM_110  ; offset+_vert_posiz_attesa_su_deposito_pinza1, quota_verticale_rulliera_prelievo_pinza1
AND>SL(323) DM_56 DM_44  ; memoria_ultimo_prelievo_pinza1, offset-_vert_posiz_attesa_su_deposito_pinza1
-L(411) DM_56 DM_62 DM_58  ; memoria_ultimo_prelievo_pinza1, step_salita_pinza1, quota_verticale_salita_dopo_prelievo_pinza1
-L(411) DM_44 DM_62 DM_60  ; offset-_vert_posiz_attesa_su_deposito_pinza1, step_salita_pinza1, quota_verticale_salita_dopo_deposito_pinza1
; rung 16: condizioni di reset quote variabili
@LD W_4003  ; stato_automatico
LDNOT W_108  ; st_pinza_1_ftc_fermata_polmone_8_prelievo_pinza_1.
ANDNOT W_6500  ; salita_dopo_prelievo_piastrella_pinza1
ORLD
MOVL(498) DM_62 DM_56  ; step_salita_pinza1, memoria_ultimo_prelievo_pinza1

### Section quote_pinza_pallet

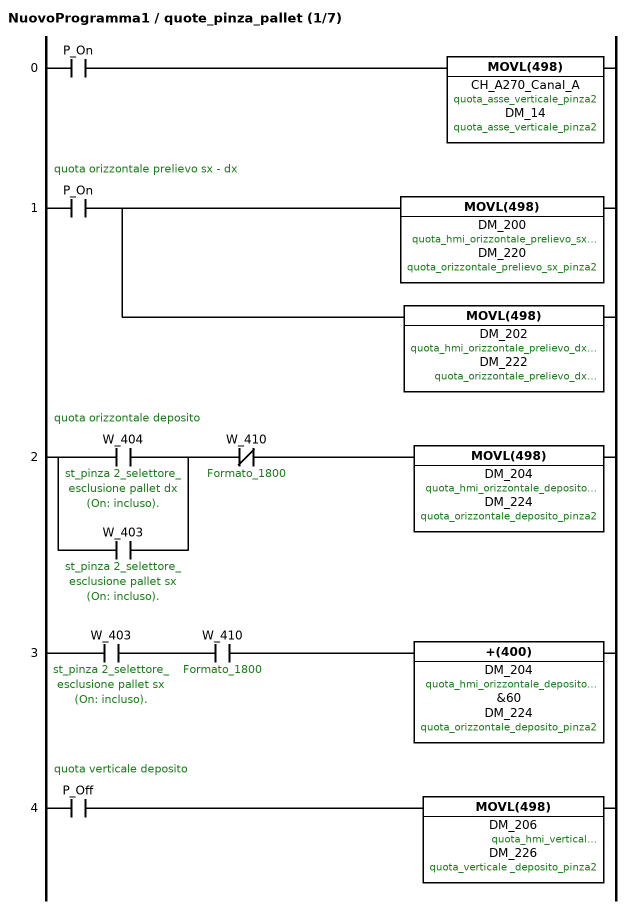
; rung 0
LD P_On
MOVL(498) CH_A270_Canal_A DM_14  ; quota_asse_verticale_pinza2
; rung 1: quota orizzontale prelievo sx - dx
LD P_On
MOVL(498) DM_200 DM_220  ; quota_hmi_orizzontale_prelievo_sx_pinza2, quota_orizzontale_prelievo_sx_pinza2
MOVL(498) DM_202 DM_222  ; quota_hmi_orizzontale_prelievo_dx_pinza2, quota_orizzontale_prelievo_dx_pinza2
; rung 2: quota orizzontale deposito
LD W_404  ; st_pinza 2_selettore_esclusione pallet dx (On: incluso).
OR W_403  ; st_pinza 2_selettore_esclusione pallet sx (On: incluso).
ANDNOT W_410  ; Formato_1800
MOVL(498) DM_204 DM_224  ; quota_hmi_orizzontale_deposito_pinza2, quota_orizzontale_deposito_pinza2
; rung 3
LD W_403  ; st_pinza 2_selettore_esclusione pallet sx (On: incluso).
AND W_410  ; Formato_1800
+(400) DM_204 &60 DM_224  ; quota_hmi_orizzontale_deposito_pinza2, quota_orizzontale_deposito_pinza2
; rung 4: quota verticale deposito
LD P_Off
MOVL(498) DM_206 DM_226  ; quota_hmi_verticale _deposito_pinza2, quota_verticale _deposito_pinza2

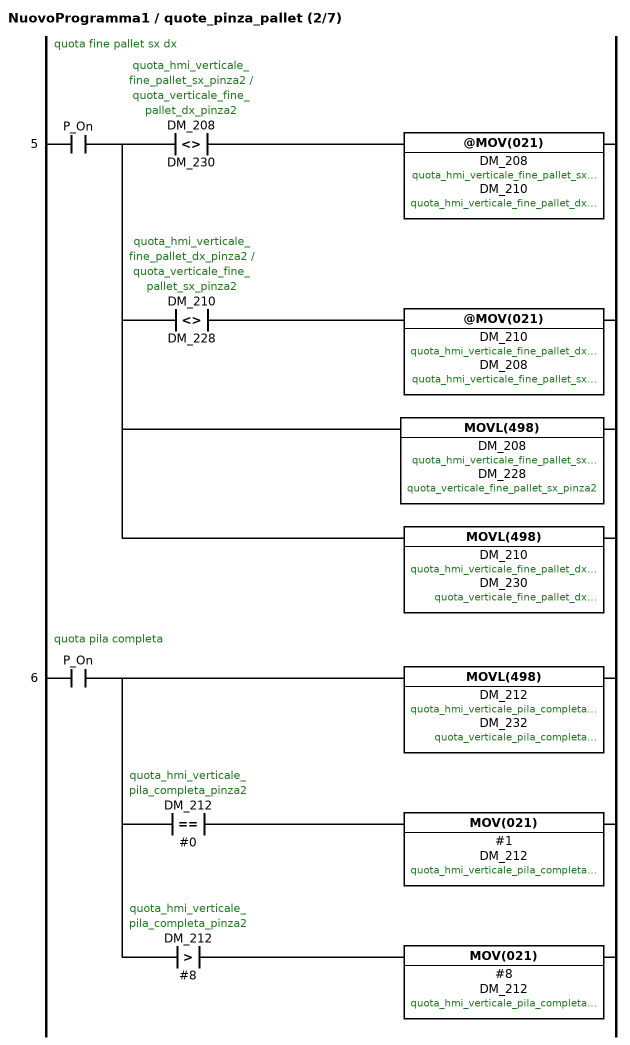
; rung 5: quota fine pallet sx dx
LD P_On
OUT TR0
AND<>(305) DM_208 DM_230  ; quota_hmi_verticale_fine_pallet_sx_pinza2, quota_verticale_fine_pallet_dx_pinza2
@MOV(021) DM_208 DM_210  ; quota_hmi_verticale_fine_pallet_sx_pinza2, quota_hmi_verticale_fine_pallet_dx_pinza2
LD TR0
AND<>(305) DM_210 DM_228  ; quota_hmi_verticale_fine_pallet_dx_pinza2, quota_verticale_fine_pallet_sx_pinza2
@MOV(021) DM_210 DM_208  ; quota_hmi_verticale_fine_pallet_dx_pinza2, quota_hmi_verticale_fine_pallet_sx_pinza2
LD TR0
MOVL(498) DM_208 DM_228  ; quota_hmi_verticale_fine_pallet_sx_pinza2, quota_verticale_fine_pallet_sx_pinza2
MOVL(498) DM_210 DM_230  ; quota_hmi_verticale_fine_pallet_dx_pinza2, quota_verticale_fine_pallet_dx_pinza2
; rung 6: quota pila completa
LD P_On
OUT TR0
MOVL(498) DM_212 DM_232  ; quota_hmi_verticale_pila_completa_pinza2, quota_verticale_pila_completa_pinza2
AND=(300) DM_212 #0  ; quota_hmi_verticale_pila_completa_pinza2
MOV(021) #1 DM_212  ; quota_hmi_verticale_pila_completa_pinza2
LD TR0
AND>(320) DM_212 #8  ; quota_hmi_verticale_pila_completa_pinza2
MOV(021) #8 DM_212  ; quota_hmi_verticale_pila_completa_pinza2

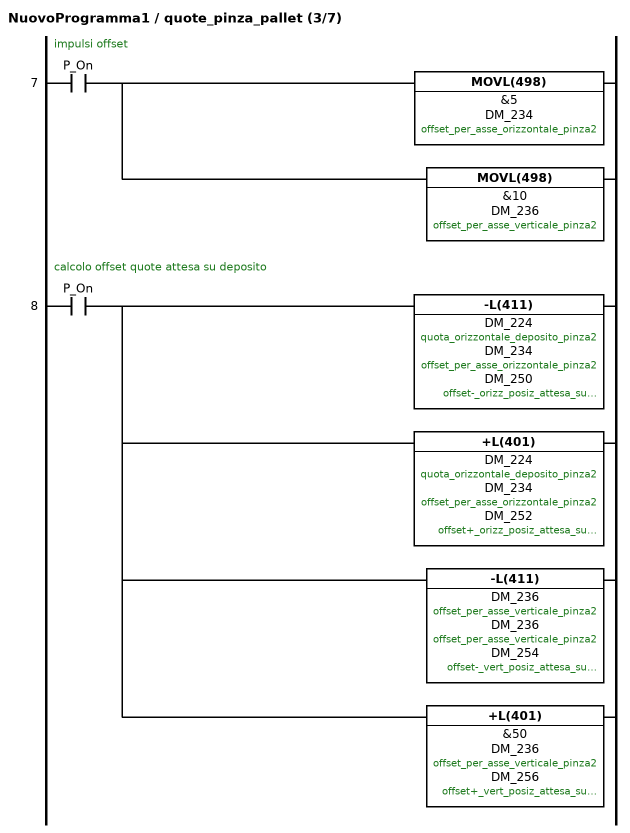
; rung 7: impulsi offset
LD P_On
MOVL(498) &5 DM_234  ; offset_per_asse_orizzontale_pinza2
MOVL(498) &10 DM_236  ; offset_per_asse_verticale_pinza2  // MOVL: Vl
; rung 8: calcolo offset quote attesa su deposito
LD P_On
-L(411) DM_224 DM_234 DM_250  ; quota_orizzontale_deposito_pinza2, offset_per_asse_orizzontale_pinza2, offset-_orizz_posiz_attesa_su_deposito_pinza2
+L(401) DM_224 DM_234 DM_252  ; quota_orizzontale_deposito_pinza2, offset_per_asse_orizzontale_pinza2, offset+_orizz_posiz_attesa_su_deposito_pinza2
-L(411) DM_236 DM_236 DM_254  ; offset_per_asse_verticale_pinza2, offset-_vert_posiz_attesa_su_deposito_pinza2
+L(401) &50 DM_236 DM_256  ; offset_per_asse_verticale_pinza2, offset+_vert_posiz_attesa_su_deposito_pinza2

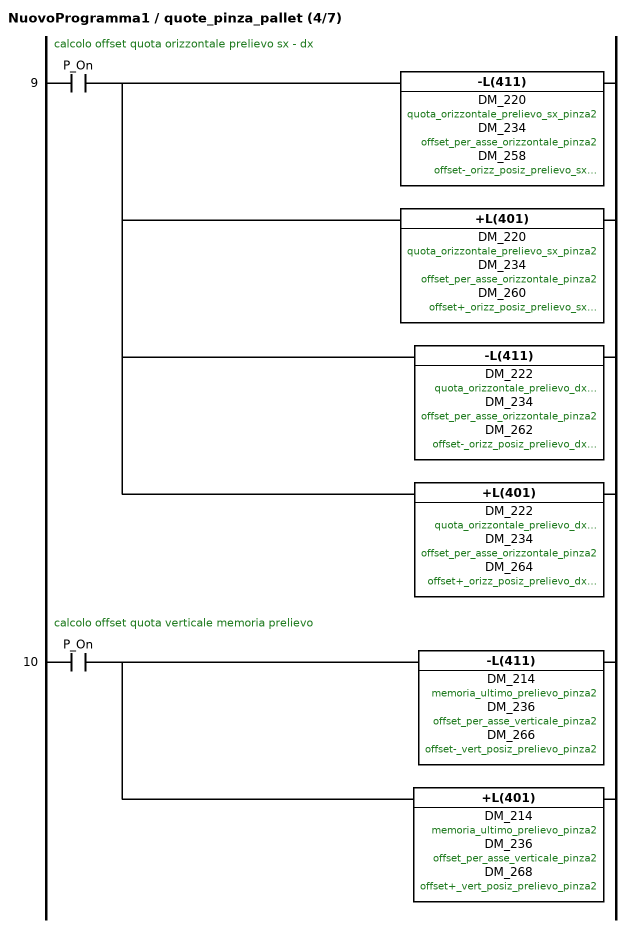
; rung 9: calcolo offset quota orizzontale prelievo sx - dx
LD P_On
-L(411) DM_220 DM_234 DM_258  ; quota_orizzontale_prelievo_sx_pinza2, offset_per_asse_orizzontale_pinza2, offset-_orizz_posiz_prelievo_sx_pinza2
+L(401) DM_220 DM_234 DM_260  ; quota_orizzontale_prelievo_sx_pinza2, offset_per_asse_orizzontale_pinza2, offset+_orizz_posiz_prelievo_sx_pinza2
-L(411) DM_222 DM_234 DM_262  ; quota_orizzontale_prelievo_dx_pinza2, offset_per_asse_orizzontale_pinza2, offset-_orizz_posiz_prelievo_dx_pinza2
+L(401) DM_222 DM_234 DM_264  ; quota_orizzontale_prelievo_dx_pinza2, offset_per_asse_orizzontale_pinza2, offset+_orizz_posiz_prelievo_dx_pinza2
; rung 10: calcolo offset quota verticale memoria prelievo
LD P_On
-L(411) DM_214 DM_236 DM_266  ; memoria_ultimo_prelievo_pinza2, offset_per_asse_verticale_pinza2, offset-_vert_posiz_prelievo_pinza2
+L(401) DM_214 DM_236 DM_268  ; memoria_ultimo_prelievo_pinza2, offset_per_asse_verticale_pinza2, offset+_vert_posiz_prelievo_pinza2

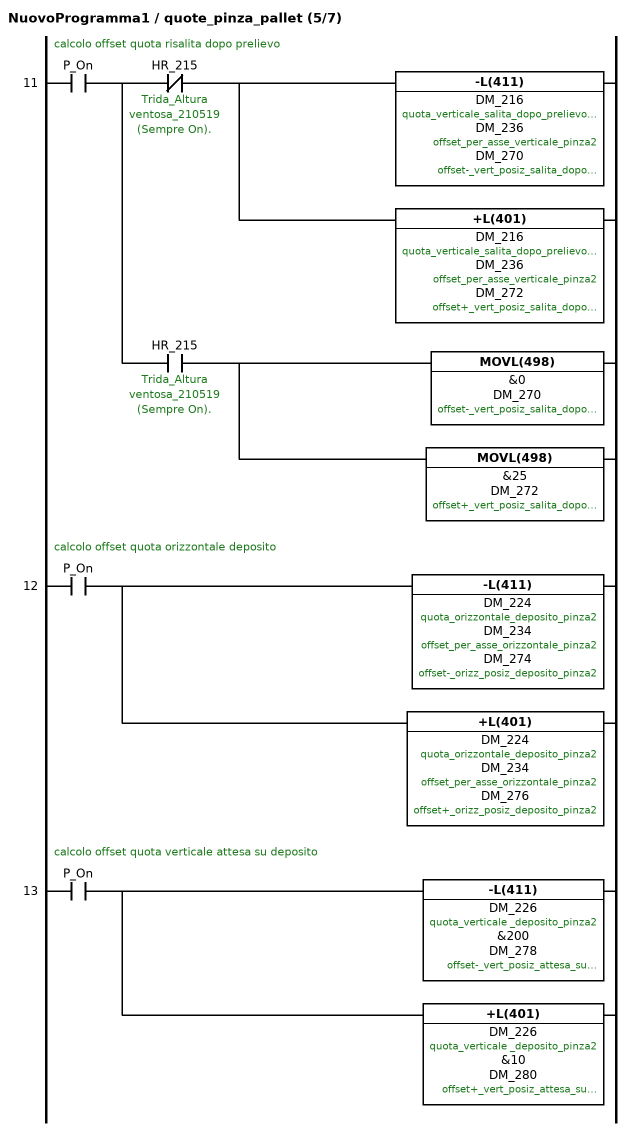
; rung 11: calcolo offset quota risalita dopo prelievo
LD P_On
OUT TR0
ANDNOT HR_215  ; Trida_Altura ventosa_210519 (Sempre On).  // H2.15: Modificado para ventosa trabalhar sempre na mesma altura. Evita problemas com pancones alto/baixo. / 210519. / .
-L(411) DM_216 DM_236 DM_270  ; quota_verticale_salita_dopo_prelievo_pinza2, offset_per_asse_verticale_pinza2, offset-_vert_posiz_salita_dopo_prelievo_pinza2
+L(401) DM_216 DM_236 DM_272  ; quota_verticale_salita_dopo_prelievo_pinza2, offset_per_asse_verticale_pinza2, offset+_vert_posiz_salita_dopo_prelievo_pinza2
LD TR0
AND HR_215  ; Trida_Altura ventosa_210519 (Sempre On).  // H2.15: Modificado para ventosa trabalhar sempre na mesma altura. Evita problemas com pancones alto/baixo. / 210519. / .
MOVL(498) &0 DM_270  ; offset-_vert_posiz_salita_dopo_prelievo_pinza2  // OBS: DM 270 sempre MENOR que Dm 272. / .
MOVL(498) &25 DM_272  ; offset+_vert_posiz_salita_dopo_prelievo_pinza2  // OBS: DM 272 sempre MAIOR que Dm 270. / .
; rung 12: calcolo offset quota orizzontale deposito
LD P_On
-L(411) DM_224 DM_234 DM_274  ; quota_orizzontale_deposito_pinza2, offset_per_asse_orizzontale_pinza2, offset-_orizz_posiz_deposito_pinza2
+L(401) DM_224 DM_234 DM_276  ; quota_orizzontale_deposito_pinza2, offset_per_asse_orizzontale_pinza2, offset+_orizz_posiz_deposito_pinza2
; rung 13: calcolo offset quota verticale attesa su deposito
LD P_On
-L(411) DM_226 &200 DM_278  ; quota_verticale _deposito_pinza2, offset-_vert_posiz_attesa_su_deposito_pinza2
+L(401) DM_226 &10 DM_280  ; quota_verticale _deposito_pinza2, offset+_vert_posiz_attesa_su_deposito_pinza2

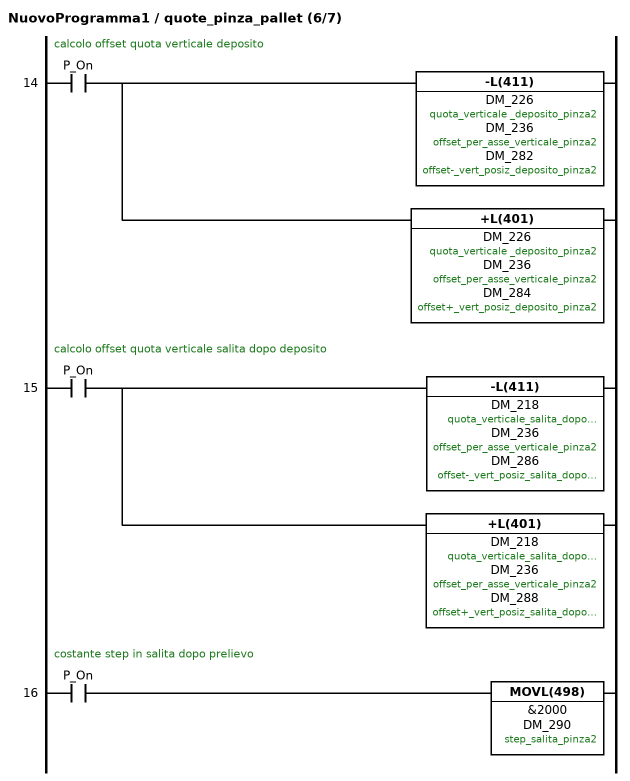
; rung 14: calcolo offset quota verticale deposito
LD P_On
-L(411) DM_226 DM_236 DM_282  ; quota_verticale _deposito_pinza2, offset_per_asse_verticale_pinza2, offset-_vert_posiz_deposito_pinza2
+L(401) DM_226 DM_236 DM_284  ; quota_verticale _deposito_pinza2, offset_per_asse_verticale_pinza2, offset+_vert_posiz_deposito_pinza2
; rung 15: calcolo offset quota verticale salita dopo deposito
LD P_On
-L(411) DM_218 DM_236 DM_286  ; quota_verticale_salita_dopo_deposito_pinza2, offset_per_asse_verticale_pinza2, offset-_vert_posiz_salita_dopo_deposito_pinza2
+L(401) DM_218 DM_236 DM_288  ; quota_verticale_salita_dopo_deposito_pinza2, offset_per_asse_verticale_pinza2, offset+_vert_posiz_salita_dopo_deposito_pinza2
; rung 16: costante step in salita dopo prelievo
LD P_On
MOVL(498) &2000 DM_290  ; step_salita_pinza2

